Yaskawa INFORM job: aruba_21-06-23_planes_program.JBI

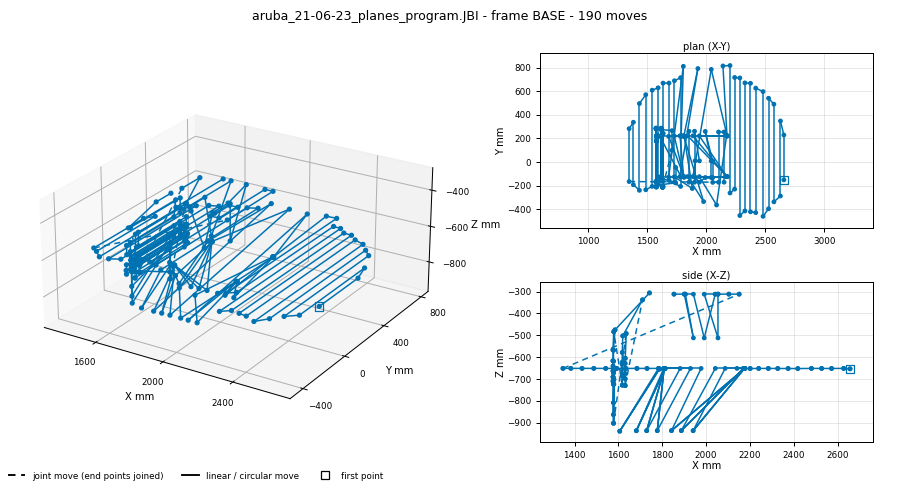
[picture p0: tool path of aruba_21-06-23_planes_program.JBI in frame BASE, 190 of 196 moves have a stored position in this frame; points joined in program order, loops and branches not executed]
/JOB
//NAME aruba_21-06-23_planes_program
//POS
///NPOS 190,0,190,0,0,0
///TOOL 0
///POSTYPE BASE
///RECTAN
///RCONF 0,0,0,0,0,0,0,0,0,0,0,0,0,0,0,0,0,0,0,0,0,0,0,0
C00000=2656.460943,-150.468551,-653.252380,175.000000,-8.848606,5.000000
C00001=2656.460943,229.117449,-653.252380,175.000000,-8.848606,5.000000
C00002=2627.497779,347.931768,-651.232478,-175.000000,-5.000000,-5.000000
C00003=2627.497779,-287.285232,-651.232478,-175.000000,-5.000000,-5.000000
C00004=2572.213711,-336.742338,-651.659154,-175.000000,-5.000000,-5.000000
C00005=2572.213711,489.916662,-651.659154,-175.000000,-5.000000,-5.000000
C00006=2526.904847,540.049866,-651.501485,-175.000000,-5.000000,-5.000000
C00007=2526.904847,-395.156134,-651.501485,-175.000000,-5.000000,-5.000000
C00008=2480.339516,-459.512372,-651.235306,-175.000000,-5.000000,-5.000000
C00009=2480.339516,596.519628,-651.235306,-175.000000,-5.000000,-5.000000
C00010=2418.281304,625.734905,-652.044532,-175.000000,-5.429419,-5.000000
C00011=2418.281304,-428.059095,-652.044532,-175.000000,-5.429419,-5.000000
C00012=2373.921678,-420.787294,-651.674768,-175.000000,-5.000000,-5.000000
C00013=2373.921678,666.630706,-651.674768,-175.000000,-5.000000,-5.000000
C00014=2326.756346,670.269706,-651.689889,-175.000000,-5.000000,-5.000000
C00015=2326.756346,-413.993294,-651.689889,-175.000000,-5.000000,-5.000000
C00016=2283.654656,-452.713368,-651.426872,-175.000000,-5.000000,-5.000000
C00017=2283.654656,712.102632,-651.426872,-175.000000,-5.000000,-5.000000
C00018=2239.829565,716.054342,-651.464834,-175.000000,5.000000,5.000000
C00019=2239.829565,-229.216658,-651.464834,-175.000000,5.000000,5.000000
C00020=2200.763302,-261.900680,-651.775326,-175.000000,5.000000,5.000000
C00021=2200.763302,817.076320,-651.775326,-175.000000,5.000000,5.000000
C00022=2140.753719,813.469514,-651.286785,-175.000000,5.000000,5.000000
C00023=2175.323719,221.429514,-651.286335,-175.000000,5.000000,5.000000
C00024=2175.323719,221.429514,-651.286335,-175.000000,5.000000,5.000000
C00025=1940.753719,221.429621,-935.816732,180.000000,-60.000000,0.000000
C00026=2174.923719,-123.582486,-651.286335,-175.000000,5.000000,5.000000
C00027=2174.923719,-123.582486,-651.286335,-175.000000,5.000000,5.000000
C00028=1940.753719,-123.582385,-935.816732,180.000000,-60.000000,0.000000
C00029=2086.834012,-363.411004,-651.203375,-175.000000,-5.000000,-5.000000
C00030=2171.404012,222.215996,-651.202925,-175.000000,-5.000000,-5.000000
C00031=2171.404012,222.215996,-651.202925,-175.000000,-5.000000,-5.000000
C00032=1886.834012,222.216104,-935.733321,180.000000,-60.000000,0.000000
C00033=2171.004012,-122.796004,-651.202925,-175.000000,-5.000000,-5.000000
C00034=2171.004012,-122.796004,-651.202925,-175.000000,-5.000000,-5.000000
C00035=1886.834012,-122.795903,-935.733321,180.000000,-60.000000,0.000000
C00036=2041.925770,784.352535,-651.263772,-175.000000,5.000000,5.000000
C00037=2176.495770,222.127535,-651.263322,-175.000000,5.000000,5.000000
C00038=2176.495770,222.127535,-651.263322,-175.000000,5.000000,5.000000
C00039=1841.925770,222.127642,-935.793718,180.000000,-60.000000,0.000000
C00040=2176.095770,-122.884465,-651.263322,-175.000000,5.000000,5.000000
C00041=2176.095770,-122.884465,-651.263322,-175.000000,5.000000,5.000000
C00042=1841.925770,-122.884364,-935.793718,180.000000,-60.000000,0.000000
C00043=1977.069048,-334.422188,-651.446071,-175.000000,-5.000000,-5.000000
C00044=1808.319048,222.466812,-651.445621,-175.000000,-5.000000,-5.000000
C00045=1808.319048,222.466812,-651.445621,-175.000000,-5.000000,-5.000000
C00046=1777.069048,222.466920,-935.976017,180.000000,-60.000000,0.000000
C00047=1808.219048,-122.545188,-651.445621,-175.000000,-5.000000,-5.000000
C00048=1808.219048,-122.545188,-651.445621,-175.000000,-5.000000,-5.000000
C00049=1777.069048,-122.545087,-935.976017,180.000000,-60.000000,0.000000
C00050=1928.721220,791.559852,-651.538855,-175.000000,-5.000000,-5.000000
C00051=1809.971220,220.040852,-651.538405,-175.000000,-5.000000,-5.000000
C00052=1809.971220,220.040852,-651.538405,-175.000000,-5.000000,-5.000000
C00053=1728.721220,220.040960,-936.068801,180.000000,-60.000000,0.000000
C00054=1809.871220,-124.971148,-651.538405,-175.000000,-5.000000,-5.000000
C00055=1809.871220,-124.971148,-651.538405,-175.000000,-5.000000,-5.000000
C00056=1728.721220,-124.971047,-936.068801,180.000000,-60.000000,0.000000
C00057=1881.497109,-223.621422,-651.637006,-174.947735,-5.000000,-5.000000
C00058=1812.747109,217.641578,-651.636556,-174.947735,-5.000000,-5.000000
C00059=1812.747109,217.641578,-651.636556,-174.947735,-5.000000,-5.000000
C00060=1681.497109,217.641686,-936.166952,180.000000,-60.000000,0.000000
C00061=1812.647109,-127.370422,-651.636556,-174.947735,-5.000000,-5.000000
C00062=1812.647109,-127.370422,-651.636556,-174.947735,-5.000000,-5.000000
C00063=1681.497109,-127.370321,-936.166952,180.000000,-60.000000,0.000000
C00064=1805.804854,810.162761,-653.872990,-175.000000,-9.014903,-5.000000
C00065=1787.054854,219.745761,-653.872540,-175.000000,-9.014903,-5.000000
C00066=1787.054854,219.745761,-653.872540,-175.000000,-9.014903,-5.000000
C00067=1605.804854,219.745869,-938.402936,180.000000,-60.000000,0.000000
C00068=1786.954854,-125.266239,-653.872540,-175.000000,-9.014903,-5.000000
C00069=1786.954854,-125.266239,-653.872540,-175.000000,-9.014903,-5.000000
C00070=1605.804854,-125.266138,-938.402936,180.000000,-60.000000,0.000000
C00071=1782.662478,-206.210679,-651.291834,-175.000000,-5.000000,-5.000000
C00072=1782.662478,714.069321,-651.291834,-175.000000,-5.000000,-5.000000
C00073=1730.212349,688.417773,-651.378037,-175.000000,-5.000000,-5.000000
C00074=1730.212349,-170.674227,-651.378037,-175.000000,-5.000000,-5.000000
C00075=1684.297183,-156.152654,-651.338765,-175.000000,-5.000000,-5.000000
C00076=1684.297183,668.531946,-651.338765,-175.000000,-5.000000,-5.000000
C00077=1633.833752,668.044159,-651.284531,-175.000000,-5.000000,-5.000000
C00078=1633.833752,-153.905441,-651.284531,-175.000000,-5.000000,-5.000000
C00079=1592.276618,-190.639632,-651.293083,-175.000000,5.000000,5.000000
C00080=1592.276618,628.548368,-651.293083,-175.000000,5.000000,5.000000
C00081=1541.838326,608.465241,-651.279954,-175.000000,5.000000,5.000000
C00082=1541.838326,-205.867759,-651.279954,-175.000000,5.000000,5.000000
C00083=1487.539467,-234.489098,-651.135826,-175.000000,5.000000,5.000000
C00084=1487.539467,569.973902,-651.135826,-175.000000,5.000000,5.000000
C00085=1433.792910,495.334747,-651.168011,-175.000000,-5.000000,-5.000000
C00086=1433.792910,-239.256253,-651.168011,-175.000000,-5.000000,-5.000000
C00087=1382.738925,-191.949702,-651.084748,-175.000000,-5.000000,-5.000000
C00088=1382.738925,337.025298,-651.084748,-175.000000,-5.000000,-5.000000
C00089=1346.852235,282.490527,-651.239445,-175.000000,5.000000,5.000000
C00090=1346.852235,-164.957473,-651.239445,-175.000000,5.000000,5.000000
C00091=2150.499142,-170.718890,-311.836795,-175.000000,-5.000000,-5.000000
C00092=2150.499142,254.705110,-311.836795,-175.000000,-5.000000,-5.000000
C00093=2103.679400,254.799372,-311.838353,-175.000000,5.000000,5.000000
C00094=2103.679400,-171.056628,-311.838353,-175.000000,5.000000,5.000000
C00095=2053.922199,-172.133646,-311.914010,-175.000000,5.000000,5.000000
C00096=2054.042199,-132.310646,-311.914225,-175.000000,5.000000,5.000000
C00097=2054.042199,8.405354,-311.914225,-175.000000,5.000000,5.000000
C00098=2053.922199,8.405654,-511.914010,-175.000000,5.000000,5.000000
C00099=1991.241004,259.354715,-312.077632,-175.000000,-5.000000,-5.000000
C00100=2041.361004,9.755715,-312.077848,-175.000000,-5.000000,-5.000000
C00101=2041.361004,-130.960285,-312.077848,-175.000000,-5.000000,-5.000000
C00102=1991.241004,-130.960285,-512.077632,-175.000000,-5.000000,-5.000000
C00103=1941.911808,-170.199961,-312.005490,-175.000000,-5.000000,-5.000000
C00104=1905.131808,-130.324961,-312.005706,-175.000000,-5.000000,-5.000000
C00105=1905.131808,10.391039,-312.005706,-175.000000,-5.000000,-5.000000
C00106=1941.911808,10.391339,-512.005490,-175.000000,-5.000000,-5.000000
C00107=1900.324174,260.964496,-311.813349,-175.000000,-5.000000,-5.000000
C00108=1900.324174,-170.738504,-311.813349,-175.000000,-5.000000,-5.000000
C00109=1853.284352,-170.551172,-311.825600,-175.000000,5.000000,5.000000
C00110=1853.284352,260.724828,-311.825600,-175.000000,5.000000,5.000000
C00111=1741.381590,-45.669052,-306.303009,180.000000,-89.999999,0.000000
C00112=1741.381590,-176.207052,-306.303009,180.000000,-89.999999,0.000000
C00113=1584.353544,-195.083398,-475.055618,180.000000,-89.999999,0.000000
C00114=1584.353544,230.369602,-475.055618,180.000000,-89.999999,0.000000
C00115=1577.352926,222.596301,-568.404381,180.000000,-89.999999,0.000000
C00116=1577.352926,-203.885699,-568.404381,180.000000,-89.999999,0.000000
C00117=1577.342619,-204.154645,-618.577970,180.000000,-89.999999,0.000000
C00118=1577.342619,222.705355,-618.577970,180.000000,-89.999999,0.000000
C00119=1577.184028,217.687895,-672.678435,180.000000,-89.999999,0.000000
C00120=1577.184028,-208.285505,-672.678435,180.000000,-89.999999,0.000000
C00121=1577.159099,-210.002270,-723.795090,180.000000,-89.999999,0.000000
C00122=1578.247563,-166.683270,-723.795090,180.000000,-89.999999,0.000000
C00123=1578.247563,-166.683270,-723.795090,180.000000,-89.999999,0.000000
C00124=1577.159099,-166.683378,-808.325036,180.000000,-60.000000,0.000000
C00125=1578.647563,178.328730,-723.795090,180.000000,-89.999999,0.000000
C00126=1578.647563,178.328730,-723.795090,180.000000,-89.999999,0.000000
C00127=1577.159099,178.328629,-808.325036,180.000000,-60.000000,0.000000
C00128=1577.106028,212.089598,-662.606578,180.000000,-60.000000,0.000000
C00129=1578.194492,-166.547702,-662.606578,180.000000,-60.000000,0.000000
C00130=1578.194492,-166.547702,-662.606578,180.000000,-60.000000,0.000000
C00131=1577.106028,-166.547810,-862.606578,180.000000,-60.000000,0.000000
C00132=1578.594492,178.464298,-662.606578,180.000000,-60.000000,0.000000
C00133=1578.594492,178.464298,-662.606578,180.000000,-60.000000,0.000000
C00134=1577.106028,178.464197,-862.606578,180.000000,-60.000000,0.000000
C00135=1577.407452,-212.883838,-701.853352,180.000000,-60.000000,0.000000
C00136=1578.495916,-165.712838,-701.853352,180.000000,-60.000000,0.000000
C00137=1578.495916,-165.712838,-701.853352,180.000000,-60.000000,0.000000
C00138=1577.407452,-165.712946,-901.853352,180.000000,-60.000000,0.000000
C00139=1578.895916,179.299162,-701.853352,180.000000,-60.000000,0.000000
C00140=1578.895916,179.299162,-701.853352,180.000000,-60.000000,0.000000
C00141=1577.407452,179.299061,-901.853352,180.000000,-60.000000,0.000000
C00142=1577.407452,179.299061,-901.853352,180.000000,-60.000000,0.000000
C00143=1635.269259,242.501099,-492.090717,180.000000,-89.999999,0.000000
C00144=1635.269259,-207.148901,-492.090717,180.000000,-89.999999,0.000000
C00145=1631.061349,-207.971067,-604.940000,180.000000,-89.999999,0.000000
C00146=1631.061349,240.598933,-604.940000,180.000000,-89.999999,0.000000
C00147=1630.974998,240.130895,-653.971486,180.000000,-89.999999,0.000000
C00148=1630.974998,-207.799105,-653.971486,180.000000,-89.999999,0.000000
C00149=1630.589566,-211.174713,-698.675585,180.000000,-89.999999,0.000000
C00150=1630.589566,239.035287,-698.675585,180.000000,-89.999999,0.000000
C00151=1630.374465,237.221709,-628.612012,180.000000,-60.000000,0.000000
C00152=1630.374465,-213.098291,-628.612012,180.000000,-60.000000,0.000000
C00153=1630.284358,-213.159504,-675.588090,180.000000,-60.000000,0.000000
C00154=1630.284358,236.730496,-675.588090,180.000000,-60.000000,0.000000
C00155=1630.418570,234.871039,-729.767750,180.000000,-60.000000,0.000000
C00156=1630.418570,-213.228961,-729.767750,180.000000,-60.000000,0.000000
C00157=1630.418570,-213.228961,-729.767750,180.000000,-60.000000,0.000000
C00158=1709.879320,99.983217,-337.785080,180.000000,-89.999999,0.000000
C00159=1709.879320,265.846217,-337.785080,180.000000,-89.999999,0.000000
C00160=1619.762523,275.472038,-502.616041,180.000000,-89.999999,0.000000
C00161=1619.762523,-160.131962,-502.616041,180.000000,-89.999999,0.000000
C00162=1617.419464,-158.625922,-578.294103,180.000000,-89.999999,0.000000
C00163=1617.419464,276.980078,-578.294103,180.000000,-89.999999,0.000000
C00164=1617.352670,276.615658,-632.957507,180.000000,-89.999999,0.000000
C00165=1617.352670,-158.159342,-632.957507,180.000000,-89.999999,0.000000
C00166=1617.369708,-153.446402,-686.390485,180.000000,-89.999999,0.000000
C00167=1617.369708,281.436598,-686.390485,180.000000,-89.999999,0.000000
C00168=1617.417708,281.411239,-623.243274,180.000000,-60.000000,0.000000
C00169=1617.417708,-154.047761,-623.243274,180.000000,-60.000000,0.000000
C00170=1617.499943,-149.907339,-675.747370,180.000000,-60.000000,0.000000
C00171=1617.499943,286.549561,-675.747370,180.000000,-60.000000,0.000000
C00172=1617.585020,286.293971,-727.548848,180.000000,-60.000000,0.000000
C00173=1617.585020,-150.003529,-727.548848,180.000000,-60.000000,0.000000
C00174=1617.585020,-150.003529,-727.548848,180.000000,-60.000000,0.000000
C00175=1578.421306,-168.245378,-483.669056,180.000000,-89.999999,0.000000
C00176=1578.421306,281.464622,-483.669056,180.000000,-89.999999,0.000000
C00177=1574.879780,283.169702,-566.585050,180.000000,-89.999999,0.000000
C00178=1574.879780,-166.690298,-566.585050,180.000000,-89.999999,0.000000
C00179=1574.842641,-168.914002,-616.421016,180.000000,-89.999999,0.000000
C00180=1574.842641,281.745998,-616.421016,180.000000,-89.999999,0.000000
C00181=1574.983384,284.628627,-663.353615,180.000000,-89.999999,0.000000
C00182=1574.983384,-166.191373,-663.353615,180.000000,-89.999999,0.000000
C00183=1575.131268,-166.473607,-709.989682,180.000000,-89.999999,0.000000
C00184=1575.131268,284.096393,-709.989682,180.000000,-89.999999,0.000000
C00185=1575.370368,286.027063,-641.184938,180.000000,-60.000000,0.000000
C00186=1575.370368,-165.712937,-641.184938,180.000000,-60.000000,0.000000
C00187=1575.428114,-164.136712,-690.599519,180.000000,-60.000000,0.000000
C00188=1575.428114,286.803288,-690.599519,180.000000,-60.000000,0.000000
C00189=1575.428114,286.803288,-690.599519,180.000000,-60.000000,0.000000
///POSTYPE PULSE
///PULSE
EC00000=0
EC00001=0
EC00002=0
EC00003=0
EC00004=0
EC00005=0
EC00006=0
EC00007=0
EC00008=0
EC00009=0
EC00010=0
EC00011=0
EC00012=0
EC00013=0
EC00014=0
EC00015=0
EC00016=0
EC00017=0
EC00018=0
EC00019=0
EC00020=0
EC00021=0
EC00022=0
EC00023=0
EC00024=0
EC00025=0
EC00026=0
EC00027=0
EC00028=0
EC00029=0
EC00030=0
EC00031=0
EC00032=0
EC00033=0
EC00034=0
EC00035=0
EC00036=0
EC00037=0
EC00038=0
EC00039=0
EC00040=0
EC00041=0
EC00042=0
EC00043=0
EC00044=0
EC00045=0
EC00046=0
EC00047=0
EC00048=0
EC00049=0
EC00050=0
EC00051=0
EC00052=0
EC00053=0
EC00054=0
EC00055=0
EC00056=0
EC00057=0
EC00058=0
EC00059=0
EC00060=0
EC00061=0
EC00062=0
EC00063=0
EC00064=0
EC00065=0
EC00066=0
EC00067=0
EC00068=0
EC00069=0
EC00070=0
EC00071=0
EC00072=0
EC00073=0
EC00074=0
EC00075=0
EC00076=0
EC00077=0
EC00078=0
EC00079=0
EC00080=0
EC00081=0
EC00082=0
EC00083=0
EC00084=0
EC00085=0
EC00086=0
EC00087=0
EC00088=0
EC00089=0
EC00090=0
EC00091=0
EC00092=0
EC00093=0
EC00094=0
EC00095=0
EC00096=0
EC00097=0
EC00098=0
EC00099=0
EC00100=0
EC00101=0
EC00102=0
EC00103=0
EC00104=0
EC00105=0
EC00106=0
EC00107=0
EC00108=0
EC00109=0
EC00110=0
EC00111=0
EC00112=0
EC00113=0
EC00114=0
EC00115=0
EC00116=0
EC00117=0
EC00118=0
EC00119=0
EC00120=0
EC00121=0
EC00122=0
EC00123=0
EC00124=0
EC00125=0
EC00126=0
EC00127=0
EC00128=0
EC00129=0
EC00130=0
EC00131=0
EC00132=0
EC00133=0
EC00134=0
EC00135=0
EC00136=0
EC00137=0
EC00138=0
EC00139=0
EC00140=0
EC00141=0
EC00142=92160
EC00143=92160
EC00144=92160
EC00145=92160
EC00146=92160
EC00147=92160
EC00148=92160
EC00149=92160
EC00150=92160
EC00151=92160
EC00152=92160
EC00153=92160
EC00154=92160
EC00155=92160
EC00156=92160
EC00157=184320
EC00158=184320
EC00159=184320
EC00160=184320
EC00161=184320
EC00162=184320
EC00163=184320
EC00164=184320
EC00165=184320
EC00166=184320
EC00167=184320
EC00168=184320
EC00169=184320
EC00170=184320
EC00171=184320
EC00172=184320
EC00173=184320
EC00174=276480
EC00175=276480
EC00176=276480
EC00177=276480
EC00178=276480
EC00179=276480
EC00180=276480
EC00181=276480
EC00182=276480
EC00183=276480
EC00184=276480
EC00185=276480
EC00186=276480
EC00187=276480
EC00188=276480
EC00189=368640
//INST
///DATE 2023/06/26 11:09
///ATTR SC,RW,RJ
////FRAME BASE
///GROUP1 RB1,ST1
NOP
MOVJ P009 EX000 VJ=15.00
MOVJ C00000 EC00000 VJ=15.0
CALL JOB:SPYON
MOVL C00001 EC00001 V=150.0
MOVL C00002 EC00002 V=150.0
MOVL C00003 EC00003 V=150.0
MOVL C00004 EC00004 V=150.0
MOVL C00005 EC00005 V=150.0
MOVL C00006 EC00006 V=150.0
MOVL C00007 EC00007 V=150.0
MOVL C00008 EC00008 V=150.0
MOVL C00009 EC00009 V=150.0
MOVL C00010 EC00010 V=150.0
MOVL C00011 EC00011 V=150.0
MOVL C00012 EC00012 V=150.0
MOVL C00013 EC00013 V=150.0
MOVL C00014 EC00014 V=150.0
MOVL C00015 EC00015 V=150.0
MOVL C00016 EC00016 V=150.0
MOVL C00017 EC00017 V=150.0
MOVL C00018 EC00018 V=150.0
MOVL C00019 EC00019 V=150.0
MOVL C00020 EC00020 V=150.0
MOVL C00021 EC00021 V=150.0
MOVL C00022 EC00022 V=150.0
MOVL C00023 EC00023 V=150.0
MOVL C00024 EC00024 V=150.0
MOVL C00025 EC00025 V=150.0
MOVL C00026 EC00026 V=150.0
MOVL C00027 EC00027 V=150.0
MOVL C00028 EC00028 V=150.0
MOVL C00029 EC00029 V=150.0
MOVL C00030 EC00030 V=150.0
MOVL C00031 EC00031 V=150.0
MOVL C00032 EC00032 V=150.0
MOVL C00033 EC00033 V=150.0
MOVL C00034 EC00034 V=150.0
MOVL C00035 EC00035 V=150.0
MOVL C00036 EC00036 V=150.0
MOVL C00037 EC00037 V=150.0
MOVL C00038 EC00038 V=150.0
MOVL C00039 EC00039 V=150.0
MOVL C00040 EC00040 V=150.0
MOVL C00041 EC00041 V=150.0
MOVL C00042 EC00042 V=150.0
MOVL C00043 EC00043 V=150.0
MOVL C00044 EC00044 V=150.0
MOVL C00045 EC00045 V=150.0
MOVL C00046 EC00046 V=150.0
MOVL C00047 EC00047 V=150.0
MOVL C00048 EC00048 V=150.0
MOVL C00049 EC00049 V=150.0
MOVL C00050 EC00050 V=150.0
MOVL C00051 EC00051 V=150.0
MOVL C00052 EC00052 V=150.0
MOVL C00053 EC00053 V=150.0
MOVL C00054 EC00054 V=150.0
MOVL C00055 EC00055 V=150.0
MOVL C00056 EC00056 V=150.0
MOVL C00057 EC00057 V=150.0
MOVL C00058 EC00058 V=150.0
MOVL C00059 EC00059 V=150.0
MOVL C00060 EC00060 V=150.0
MOVL C00061 EC00061 V=150.0
MOVL C00062 EC00062 V=150.0
MOVL C00063 EC00063 V=150.0
MOVL C00064 EC00064 V=150.0
MOVL C00065 EC00065 V=150.0
MOVL C00066 EC00066 V=150.0
MOVL C00067 EC00067 V=150.0
MOVL C00068 EC00068 V=150.0
MOVL C00069 EC00069 V=150.0
MOVL C00070 EC00070 V=150.0
MOVL C00071 EC00071 V=150.0
MOVL C00072 EC00072 V=150.0
MOVL C00073 EC00073 V=150.0
MOVL C00074 EC00074 V=150.0
MOVL C00075 EC00075 V=150.0
MOVL C00076 EC00076 V=150.0
MOVL C00077 EC00077 V=150.0
MOVL C00078 EC00078 V=150.0
MOVL C00079 EC00079 V=150.0
MOVL C00080 EC00080 V=150.0
MOVL C00081 EC00081 V=150.0
MOVL C00082 EC00082 V=150.0
MOVL C00083 EC00083 V=150.0
MOVL C00084 EC00084 V=150.0
MOVL C00085 EC00085 V=150.0
MOVL C00086 EC00086 V=150.0
MOVL C00087 EC00087 V=150.0
MOVL C00088 EC00088 V=150.0
MOVL C00089 EC00089 V=150.0
MOVL C00090 EC00090 V=150.0
CALL JOB:SPYOF
MOVJ C00091 EC00091 VJ=15.0
CALL JOB:SPYON
MOVL C00092 EC00092 V=150.0
MOVL C00093 EC00093 V=150.0
MOVL C00094 EC00094 V=150.0
MOVL C00095 EC00095 V=150.0
MOVL C00096 EC00096 V=150.0
MOVL C00097 EC00097 V=150.0
MOVL C00098 EC00098 V=150.0
MOVL C00099 EC00099 V=150.0
MOVL C00100 EC00100 V=150.0
MOVL C00101 EC00101 V=150.0
MOVL C00102 EC00102 V=150.0
MOVL C00103 EC00103 V=150.0
MOVL C00104 EC00104 V=150.0
MOVL C00105 EC00105 V=150.0
MOVL C00106 EC00106 V=150.0
MOVL C00107 EC00107 V=150.0
MOVL C00108 EC00108 V=150.0
MOVL C00109 EC00109 V=150.0
MOVL C00110 EC00110 V=150.0
CALL JOB:SPYOF
MOVJ P009 VJ=15.00
MOVJ C00111 EC00111 VJ=15.0
CALL JOB:SPYON
MOVL C00112 EC00112 V=150.0
MOVL C00113 EC00113 V=150.0
MOVL C00114 EC00114 V=150.0
MOVL C00115 EC00115 V=150.0
MOVL C00116 EC00116 V=150.0
MOVL C00117 EC00117 V=150.0
MOVL C00118 EC00118 V=150.0
MOVL C00119 EC00119 V=150.0
MOVL C00120 EC00120 V=150.0
MOVL C00121 EC00121 V=150.0
MOVL C00122 EC00122 V=150.0
MOVL C00123 EC00123 V=150.0
MOVL C00124 EC00124 V=150.0
MOVL C00125 EC00125 V=150.0
MOVL C00126 EC00126 V=150.0
MOVL C00127 EC00127 V=150.0
MOVL C00128 EC00128 V=150.0
MOVL C00129 EC00129 V=150.0
MOVL C00130 EC00130 V=150.0
MOVL C00131 EC00131 V=150.0
MOVL C00132 EC00132 V=150.0
MOVL C00133 EC00133 V=150.0
MOVL C00134 EC00134 V=150.0
MOVL C00135 EC00135 V=150.0
MOVL C00136 EC00136 V=150.0
MOVL C00137 EC00137 V=150.0
MOVL C00138 EC00138 V=150.0
MOVL C00139 EC00139 V=150.0
MOVL C00140 EC00140 V=150.0
MOVL C00141 EC00141 V=150.0
CALL JOB:SPYOF
MOVJ P009 VJ=15.00
MOVL C00142 EC00142 V=150.0
MOVJ C00143 EC00143 VJ=15.0
CALL JOB:SPYON
MOVL C00144 EC00144 V=150.0
MOVL C00145 EC00145 V=150.0
MOVL C00146 EC00146 V=150.0
MOVL C00147 EC00147 V=150.0
MOVL C00148 EC00148 V=150.0
MOVL C00149 EC00149 V=150.0
MOVL C00150 EC00150 V=150.0
MOVL C00151 EC00151 V=150.0
MOVL C00152 EC00152 V=150.0
MOVL C00153 EC00153 V=150.0
MOVL C00154 EC00154 V=150.0
MOVL C00155 EC00155 V=150.0
MOVL C00156 EC00156 V=150.0
CALL JOB:SPYOF
MOVJ P009 VJ=15.00
MOVL C00157 EC00157 V=150.0
MOVJ C00158 EC00158 VJ=15.0
CALL JOB:SPYON
MOVL C00159 EC00159 V=150.0
MOVL C00160 EC00160 V=150.0
MOVL C00161 EC00161 V=150.0
MOVL C00162 EC00162 V=150.0
MOVL C00163 EC00163 V=150.0
MOVL C00164 EC00164 V=150.0
MOVL C00165 EC00165 V=150.0
MOVL C00166 EC00166 V=150.0
MOVL C00167 EC00167 V=150.0
MOVL C00168 EC00168 V=150.0
MOVL C00169 EC00169 V=150.0
MOVL C00170 EC00170 V=150.0
MOVL C00171 EC00171 V=150.0
MOVL C00172 EC00172 V=150.0
MOVL C00173 EC00173 V=150.0
CALL JOB:SPYOF
MOVJ P009 VJ=15.00
MOVL C00174 EC00174 V=150.0
MOVJ C00175 EC00175 VJ=15.0
CALL JOB:SPYON
MOVL C00176 EC00176 V=150.0
MOVL C00177 EC00177 V=150.0
MOVL C00178 EC00178 V=150.0
MOVL C00179 EC00179 V=150.0
MOVL C00180 EC00180 V=150.0
MOVL C00181 EC00181 V=150.0
MOVL C00182 EC00182 V=150.0
MOVL C00183 EC00183 V=150.0
MOVL C00184 EC00184 V=150.0
MOVL C00185 EC00185 V=150.0
MOVL C00186 EC00186 V=150.0
MOVL C00187 EC00187 V=150.0
MOVL C00188 EC00188 V=150.0
CALL JOB:SPYOF
MOVJ P009 VJ=15.00
MOVL C00189 EC00189 V=150.0
END
